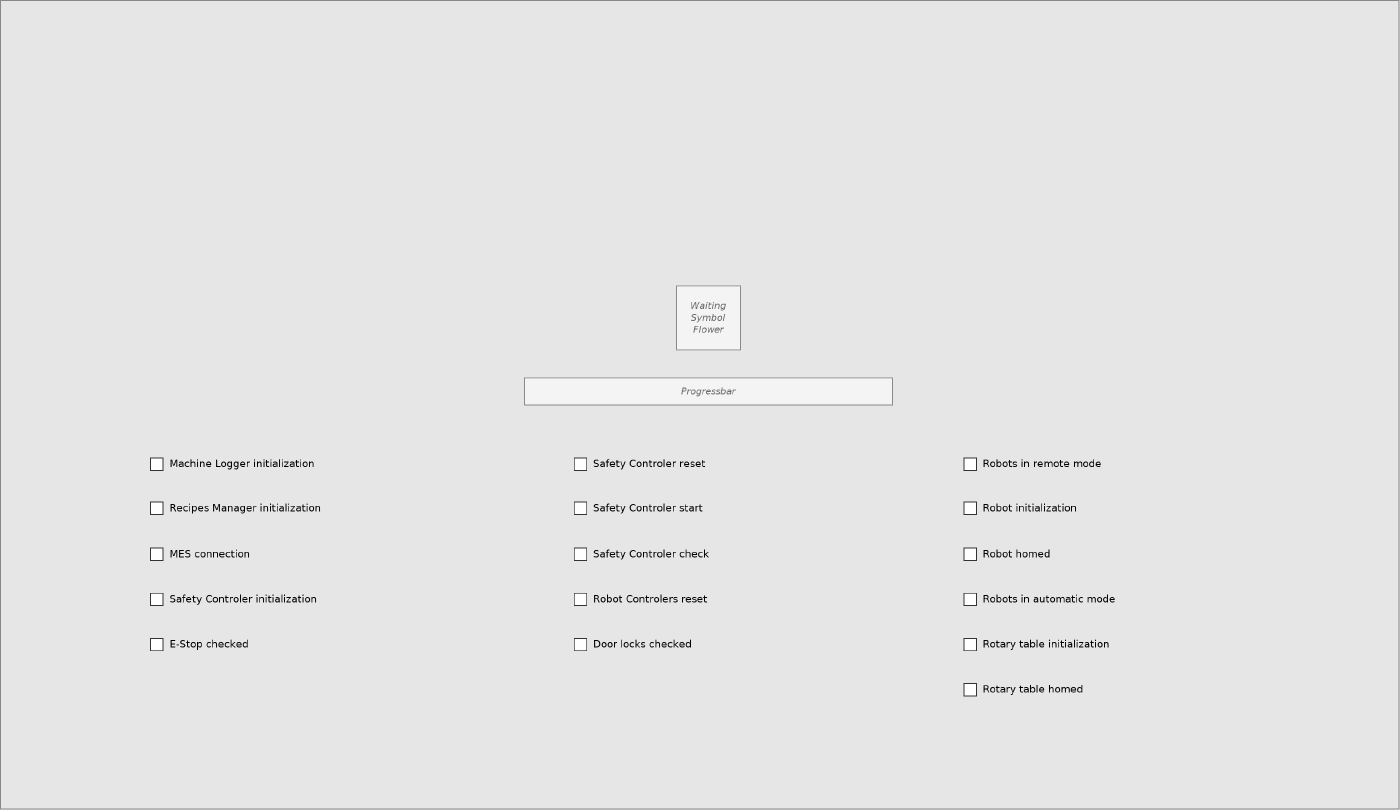
VISUALIZATION PageInitializing  // 1520x880
VAR_IN_OUT
	iProgressBar : USINT;
END_VAR
    Progressbar (569,410 400x30), variable: iProgressBar
    WaitingSymbolFlower (734,310 70x70)
    Checkbox (161,489 300x30), "Machine Logger initialization", variable: PRG_VisuControl.fbVisuControl.stInitializingFrame.bMachineLoggerInitialized, input disabled if: FALSE
    Checkbox (621,636 320x30), "Robot Controlers reset", variable: PRG_VisuControl.fbVisuControl.stInitializingFrame.bRobotControlersResetDone
    Checkbox (1044,537 320x30), "Robot initialization", variable: PRG_VisuControl.fbVisuControl.stInitializingFrame.bRobotOneInitialized
    Checkbox (1044,636 300x30), "Robots in automatic mode", variable: PRG_VisuControl.fbVisuControl.stInitializingFrame.bRobotsInAutomaticMode
    Checkbox (1044,587 320x30), "Robot homed", variable: PRG_VisuControl.fbVisuControl.stInitializingFrame.bRobotOneHomed
    Checkbox (161,537 300x30), "Recipes Manager initialization", variable: PRG_VisuControl.fbVisuControl.stInitializingFrame.bRecipesManagerInitialized, input disabled if: FALSE
    Checkbox (161,587 300x30), "MES connection", variable: PRG_VisuControl.fbVisuControl.stInitializingFrame.bMesConnected, input disabled if: FALSE
    Checkbox (161,636 300x30), "Safety Controler initialization", variable: PRG_VisuControl.fbVisuControl.stInitializingFrame.bSafetyInitialization, input disabled if: FALSE
    Checkbox (161,685 300x30), "E-Stop checked", variable: PRG_VisuControl.fbVisuControl.stInitializingFrame.bEStopChecked, input disabled if: FALSE
    Checkbox (621,685 300x30), "Door locks checked", variable: PRG_VisuControl.fbVisuControl.stInitializingFrame.bDoorsLocked, input disabled if: FALSE
    Checkbox (621,489 320x30), "Safety Controler reset", variable: PRG_VisuControl.fbVisuControl.stInitializingFrame.bSafetyReset, input disabled if: FALSE
    Checkbox (621,537 320x30), "Safety Controler start", variable: PRG_VisuControl.fbVisuControl.stInitializingFrame.bSafetyStart, input disabled if: FALSE
    Checkbox (621,587 320x30), "Safety Controler check", variable: PRG_VisuControl.fbVisuControl.stInitializingFrame.bSafetyCheck
    Checkbox (1044,489 320x30), "Robots in remote mode", variable: PRG_VisuControl.fbVisuControl.stInitializingFrame.bRobotsInRemoteMode
    Checkbox (1044,734 208x30), "Rotary table homed"
    Checkbox (1044,685 293x30), "Rotary table initialization"
END_VISUALIZATION

(* stored: Version 1.1.0.1, ProductVersion 3.1.4024.9
   Visu PageInitializing: Id {461aef6d-9bf3-405f-b92f-526b7bdc38b8} *)
